// ---- HMI1/Screens/Motion/Mot_010_Motions.TcVIS
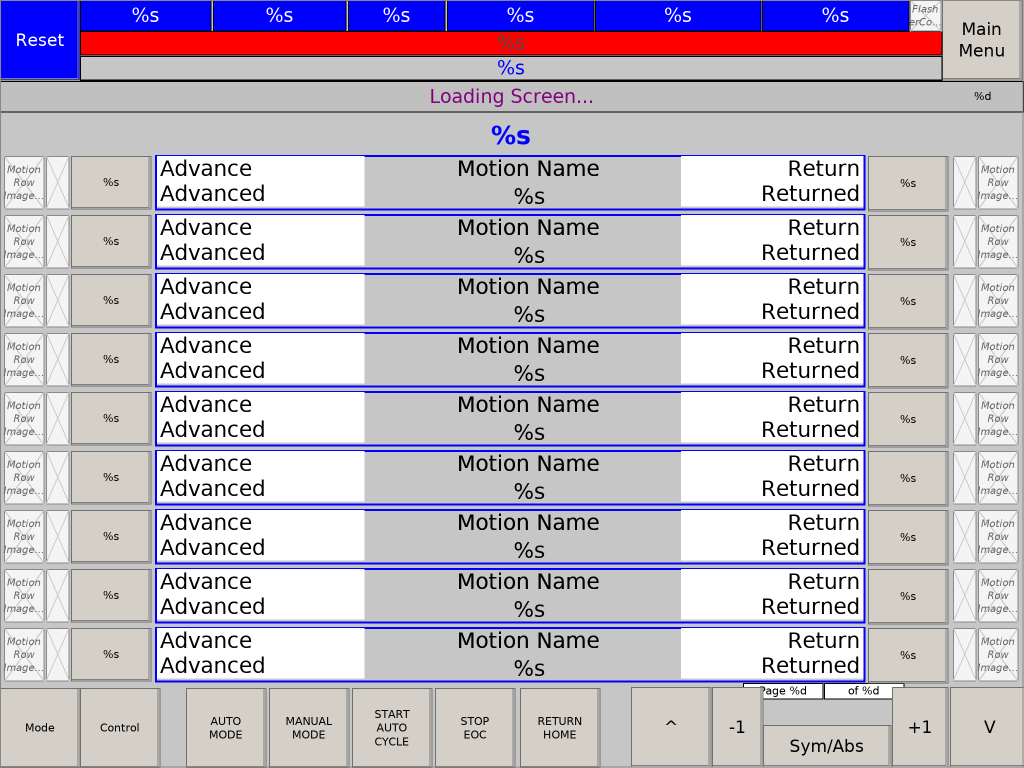
VISUALIZATION Mot_010_Motions  // 1024x768
    Frame (0,0 1024x768)
        shows Tmp_000_Template(header := gHMIData.hmiHeader)
    Frame (0,155 1024x55)
        shows MotionRow(MotionRowInstanceSingle := gHMIMotionRows.gMotionRows.gMotionRow1, MotionRowButtonsSingle := gHMIMotionRows.gMotionRowButtons.gMotionRow1btn)
    Frame (0,214 1024x55)
        shows MotionRow(MotionRowInstanceSingle := gHMIMotionRows.gMotionRows.gMotionRow2, MotionRowButtonsSingle := gHMIMotionRows.gMotionRowButtons.gMotionRow2btn)
    Frame (0,273 1024x55)
        shows MotionRow(MotionRowInstanceSingle := gHMIMotionRows.gMotionRows.gMotionRow3, MotionRowButtonsSingle := gHMIMotionRows.gMotionRowButtons.gMotionRow3btn)
    Frame (0,332 1024x55)
        shows MotionRow(MotionRowInstanceSingle := gHMIMotionRows.gMotionRows.gMotionRow4, MotionRowButtonsSingle := gHMIMotionRows.gMotionRowButtons.gMotionRow4btn)
    Frame (0,391 1024x55)
        shows MotionRow(MotionRowInstanceSingle := gHMIMotionRows.gMotionRows.gMotionRow5, MotionRowButtonsSingle := gHMIMotionRows.gMotionRowButtons.gMotionRow5btn)
    Frame (0,450 1024x55)
        shows MotionRow(MotionRowInstanceSingle := gHMIMotionRows.gMotionRows.gMotionRow6, MotionRowButtonsSingle := gHMIMotionRows.gMotionRowButtons.gMotionRow6btn)
    Button (763,725 128x42), "Sym/Abs", colour toggle: gHMIButtons.btnAbsMode
        toggle gHMIButtons.btnAbsMode
        OnMouseDown: execute { gHMIButtons.gAnyButtonPressed := TRUE; }
    Button (631,687 80x80), "^"
        tap gHMIButtons.btnPrevPage
        OnMouseDown: execute { gHMIButtons.gAnyButtonPressed := TRUE; }
    Button (950,687 80x80), "V"
        tap gHMIButtons.btnNextPage
        OnMouseDown: execute { gHMIButtons.gAnyButtonPressed := TRUE; }
    Rectangle (743,683 80x16), "Page %d", text variable: gHMIData.gActivePageNumber
        OnMouseDown: execute { gHMIButtons.gAnyButtonPressed := TRUE; }
    Rectangle (824,683 80x16), "of %d", text variable: gHMIData.gMaxPageNumber
        OnMouseDown: execute { gHMIButtons.gAnyButtonPressed := TRUE; }
    Rectangle (5,116 1012x38), "%s", text list: 'ManualPageTitle', text index: gHMIData.gManualScreenTitle
    Frame (0,509 1024x55)
        shows MotionRow(MotionRowInstanceSingle := gHMIMotionRows.gMotionRows.gMotionRow7, MotionRowButtonsSingle := gHMIMotionRows.gMotionRowButtons.gMotionRow7btn)
    Frame (0,568 1024x55)
        shows MotionRow(MotionRowInstanceSingle := gHMIMotionRows.gMotionRows.gMotionRow8, MotionRowButtonsSingle := gHMIMotionRows.gMotionRowButtons.gMotionRow8btn)
    Frame (0,627 1024x55)
        shows MotionRow(MotionRowInstanceSingle := gHMIMotionRows.gMotionRows.gMotionRow9, MotionRowButtonsSingle := gHMIMotionRows.gMotionRowButtons.gMotionRow9btn)
    Button (712,687 51x80), "-1"
        tap gHMIButtons.btnNeg1Row
        OnMouseDown: execute { gHMIButtons.gAnyButtonPressed := TRUE; }
    Button (892,687 56x80), "+1"
        tap gHMIButtons.btnPlus1Row
        OnMouseDown: execute { gHMIButtons.gAnyButtonPressed := TRUE; }
END_VISUALIZATION

// ---- HMI1/Screens/Motion/Mot_011_Axis.TcVIS
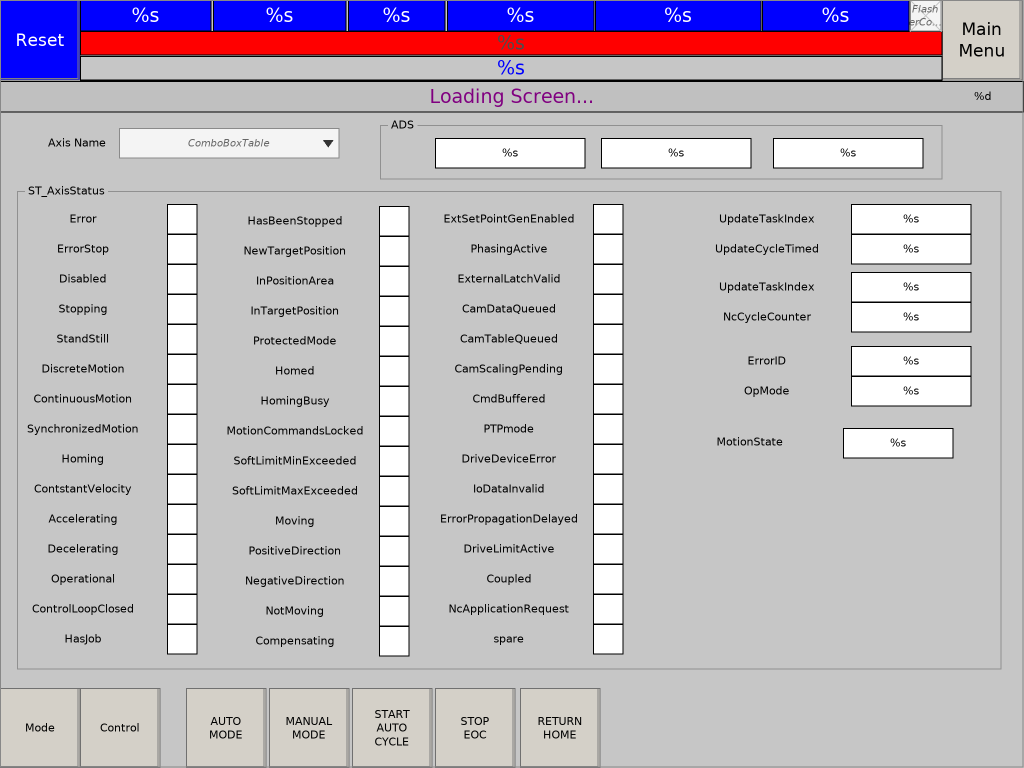
VISUALIZATION Mot_011_Axis  // 1024x768
    Frame (0,0 1024x768)
        shows Tmp_000_Template(header := gHMIData.hmiHeader)
    GroupBox (380,117 562x62), "ADS"
    GroupBox (17,183 984x486), "ST_AxisStatus"
        Label (658,244 150x30), "MotionState"
        Rectangle (826,245 110x30), "%s", text variable: driveGlobals.hmiAxis.Status.MotionState
    ComboBoxTable (119,128 220x30), variable: driveGlobals.hmiAxisSel, data array: driveGlobals.tAxisList
        p3854506369: driveGlobals.tAxisList[INDEX]
        p1128707560: Axis.gNumAxisInSystem
    Label (2,128 150x30), "Axis Name"
    Rectangle (435,138 150x30), "%s", text variable: driveGlobals.hmiAxis.ADS.Channel
    Rectangle (601,138 150x30), "%s", text variable: driveGlobals.hmiAxis.ADS.NetId
    Rectangle (773,138 150x30), "%s", text variable: driveGlobals.hmiAxis.ADS.Port
    Label (8,204 150x30), "Error"
    Rectangle (167,204 30x30), colour toggle: driveGlobals.hmiAxis.Status.Error
    Label (8,234 150x30), "ErrorStop"
    Rectangle (167,234 30x30), colour toggle: driveGlobals.hmiAxis.Status.ErrorStop
    Label (8,264 150x30), "Disabled"
    Rectangle (167,264 30x30), colour toggle: driveGlobals.hmiAxis.Status.Disabled
    Label (8,294 150x30), "Stopping"
    Rectangle (167,294 30x30), colour toggle: driveGlobals.hmiAxis.Status.Stopping
    Label (8,324 150x30), "StandStill"
    Rectangle (167,324 30x30), colour toggle: driveGlobals.hmiAxis.Status.StandStill
    Label (8,354 150x30), "DiscreteMotion"
    Rectangle (167,354 30x30), colour toggle: driveGlobals.hmiAxis.Status.DiscreteMotion
    Label (8,384 150x30), "ContinuousMotion"
    Rectangle (167,384 30x30), colour toggle: driveGlobals.hmiAxis.Status.ContinuousMotion
    Label (8,414 150x30), "SynchronizedMotion"
    Rectangle (167,414 30x30), colour toggle: driveGlobals.hmiAxis.Status.SynchronizedMotion
    Label (8,444 150x30), "Homing"
    Rectangle (167,444 30x30), colour toggle: driveGlobals.hmiAxis.Status.Homing
    Label (8,474 150x30), "ContstantVelocity"
    Rectangle (167,474 30x30), colour toggle: driveGlobals.hmiAxis.Status.ConstantVelocity
    Label (8,504 150x30), "Accelerating"
    Rectangle (167,504 30x30), colour toggle: driveGlobals.hmiAxis.Status.Accelerating
    Label (8,534 150x30), "Decelerating"
    Rectangle (167,534 30x30), colour toggle: driveGlobals.hmiAxis.Status.Decelerating
    Label (8,564 150x30), "Operational"
    Rectangle (167,564 30x30), colour toggle: driveGlobals.hmiAxis.Status.Operational
    Label (8,594 150x30), "ControlLoopClosed"
    Rectangle (167,594 30x30), colour toggle: driveGlobals.hmiAxis.Status.ControlLoopClosed
    Label (8,624 150x30), "HasJob"
    Rectangle (167,624 30x30), colour toggle: driveGlobals.hmiAxis.Status.HasJob
    Label (220,206 150x30), "HasBeenStopped"
    Rectangle (379,206 30x30), colour toggle: driveGlobals.hmiAxis.Status.HasBeenStopped
    Label (220,236 150x30), "NewTargetPosition"
    Rectangle (379,236 30x30), colour toggle: driveGlobals.hmiAxis.Status.NewTargetPosition
    Label (220,266 150x30), "InPositionArea"
    Rectangle (379,266 30x30), colour toggle: driveGlobals.hmiAxis.Status.InPositionArea
    Label (220,296 150x30), "InTargetPosition"
    Rectangle (379,296 30x30), colour toggle: driveGlobals.hmiAxis.Status.InTargetPosition
    Label (220,326 150x30), "ProtectedMode"
    Rectangle (379,326 30x30), colour toggle: driveGlobals.hmiAxis.Status.ProtectedMode
    Label (220,356 150x30), "Homed"
    Rectangle (379,356 30x30), colour toggle: driveGlobals.hmiAxis.Status.Homed
    Label (220,386 150x30), "HomingBusy"
    Rectangle (379,386 30x30), colour toggle: driveGlobals.hmiAxis.Status.HomingBusy
    Label (220,416 150x30), "MotionCommandsLocked"
    Rectangle (379,416 30x30), colour toggle: driveGlobals.hmiAxis.Status.MotionCommandsLocked
    Label (220,446 150x30), "SoftLimitMinExceeded"
    Rectangle (379,446 30x30), colour toggle: driveGlobals.hmiAxis.Status.SoftLimitMinExceeded
    Label (220,476 150x30), "SoftLimitMaxExceeded"
    Rectangle (379,476 30x30), colour toggle: driveGlobals.hmiAxis.Status.SoftLimitMaxExceeded
    Label (220,506 150x30), "Moving"
    Rectangle (379,506 30x30), colour toggle: driveGlobals.hmiAxis.Status.Moving
    Label (220,536 150x30), "PositiveDirection"
    Rectangle (379,536 30x30), colour toggle: driveGlobals.hmiAxis.Status.PositiveDirection
    Label (220,566 150x30), "NegativeDirection"
    Rectangle (379,566 30x30), colour toggle: driveGlobals.hmiAxis.Status.NegativeDirection
    Label (220,596 150x30), "NotMoving"
    Rectangle (379,596 30x30), colour toggle: driveGlobals.hmiAxis.Status.NotMoving
    Label (220,626 150x30), "Compensating"
    Rectangle (379,626 30x30), colour toggle: driveGlobals.hmiAxis.Status.Compensating
    Label (434,204 150x30), "ExtSetPointGenEnabled"
    Rectangle (593,204 30x30), colour toggle: driveGlobals.hmiAxis.Status.ExtSetPointGenEnabled
    Label (434,234 150x30), "PhasingActive"
    Rectangle (593,234 30x30), colour toggle: driveGlobals.hmiAxis.Status.PhasingActive
    Label (434,264 150x30), "ExternalLatchValid"
    Rectangle (593,264 30x30), colour toggle: driveGlobals.hmiAxis.Status.ExternalLatchValid
    Label (434,294 150x30), "CamDataQueued"
    Rectangle (593,294 30x30), colour toggle: driveGlobals.hmiAxis.Status.CamDataQueued
    Label (434,324 150x30), "CamTableQueued"
    Rectangle (593,324 30x30), colour toggle: driveGlobals.hmiAxis.Status.CamTableQueued
    Label (434,354 150x30), "CamScalingPending"
    Rectangle (593,354 30x30), colour toggle: driveGlobals.hmiAxis.Status.CamScalingPending
    Label (434,384 150x30), "CmdBuffered"
    Rectangle (593,384 30x30), colour toggle: driveGlobals.hmiAxis.Status.CmdBuffered
    Label (434,414 150x30), "PTPmode"
    Rectangle (593,414 30x30), colour toggle: driveGlobals.hmiAxis.Status.PTPmode
    Label (434,444 150x30), "DriveDeviceError"
    Rectangle (593,444 30x30), colour toggle: driveGlobals.hmiAxis.Status.DriveDeviceError
    Label (434,474 150x30), "IoDataInvalid"
    Rectangle (593,474 30x30), colour toggle: driveGlobals.hmiAxis.Status.IoDataInvalid
    Label (434,504 150x30), "ErrorPropagationDelayed"
    Rectangle (593,504 30x30), colour toggle: driveGlobals.hmiAxis.Status.ErrorPropagationDelayed
    Label (434,534 150x30), "DriveLimitActive"
    Rectangle (593,534 30x30), colour toggle: driveGlobals.hmiAxis.Status.DriveLimitActive
    Label (434,564 150x30), "Coupled"
    Rectangle (593,564 30x30), colour toggle: driveGlobals.hmiAxis.Status.Coupled
    Label (434,594 150x30), "NcApplicationRequest"
    Rectangle (593,594 30x30), colour toggle: driveGlobals.hmiAxis.Status.NcApplicationRequest
    Label (434,624 150x30), "spare"
    Rectangle (593,624 30x30)
    Label (692,204 150x30), "UpdateTaskIndex"
    Rectangle (851,204 120x30), "%s", text variable: driveGlobals.hmiAxis.Status.UpdateTaskIndex
    Label (692,234 150x30), "UpdateCycleTimed"
    Rectangle (851,234 120x30), "%s", text variable: driveGlobals.hmiAxis.Status.UpdateCycleTime
    Label (692,272 150x30), "UpdateTaskIndex"
    Rectangle (851,272 120x30), "%s"
    Label (692,302 150x30), "NcCycleCounter"
    Rectangle (851,302 120x30), "%s", text variable: driveGlobals.hmiAxis.Status.NcCycleCounter
    Label (692,346 150x30), "ErrorID"
    Rectangle (851,346 120x30), "%s", text variable: driveGlobals.hmiAxis.Status.ErrorID
    Label (692,376 150x30), "OpMode"
    Rectangle (851,376 120x30), "%s"
END_VISUALIZATION

// ---- HMI1/Screens/Popup/PopupMenu1.TcVIS
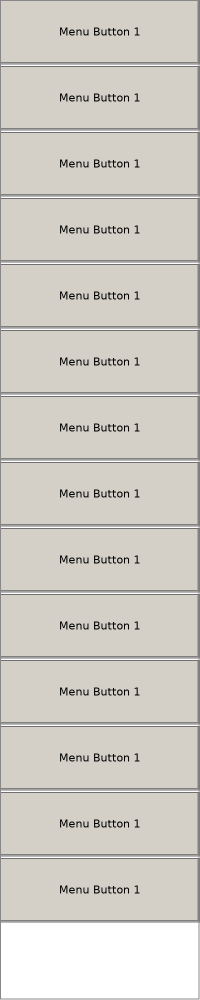
VISUALIZATION PopupMenu1  // 200x1000
    Button (0,0 200x64), "Menu Button 1"
    Button (0,66 200x64), "Menu Button 1"
    Button (0,132 200x64), "Menu Button 1"
    Button (0,198 200x64), "Menu Button 1"
    Button (0,264 200x64), "Menu Button 1"
    Button (0,330 200x64), "Menu Button 1"
    Button (0,396 200x64), "Menu Button 1"
    Button (0,462 200x64), "Menu Button 1"
    Button (0,528 200x64), "Menu Button 1"
    Button (0,594 200x64), "Menu Button 1"
    Button (0,660 200x64), "Menu Button 1"
    Button (0,726 200x64), "Menu Button 1"
    Button (0,792 200x64), "Menu Button 1"
    Button (0,858 200x64), "Menu Button 1"
END_VISUALIZATION

// ---- HMI1/Screens/Popup/PopupMenu2.TcVIS
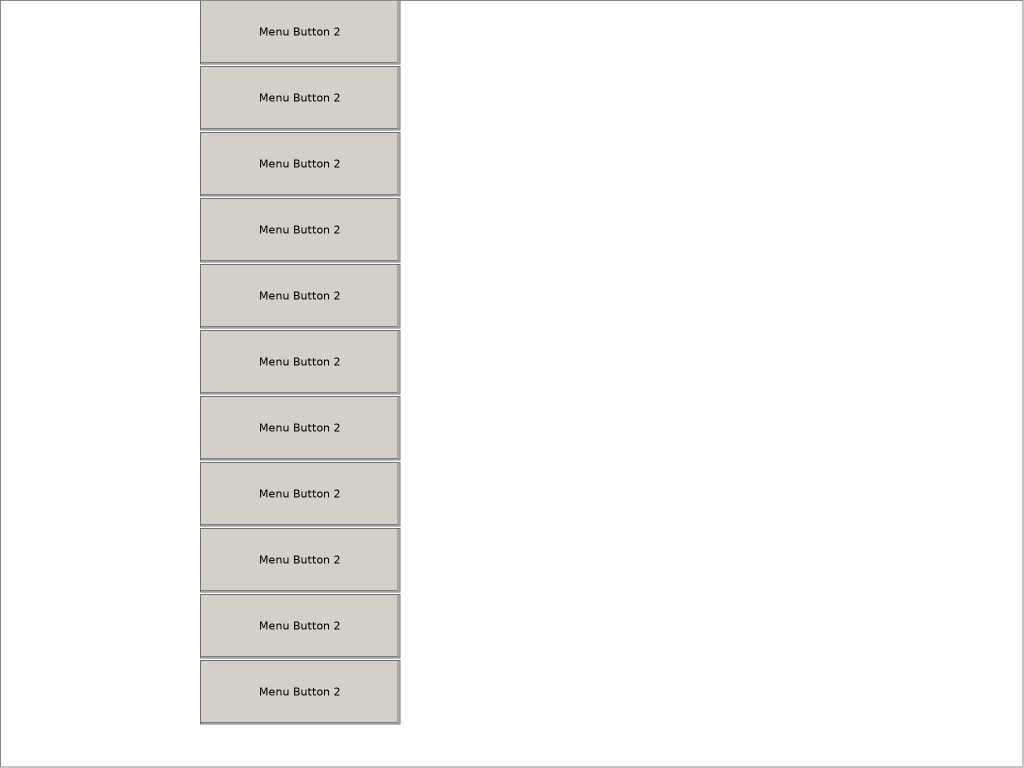
VISUALIZATION PopupMenu2  // 1024x768
    Button (200,0 200x64), "Menu Button 2"
        OnMouseClick: CloseDialog Dialog=PopupMenu2, Result=None, NumpadKeypadSet=True
    Button (200,66 200x64), "Menu Button 2"
        OnMouseClick: CloseDialog Dialog=PopupMenu2, Result=None, NumpadKeypadSet=True
    Button (200,132 200x64), "Menu Button 2"
        OnMouseClick: CloseDialog Dialog=PopupMenu2, Result=None, NumpadKeypadSet=True
    Button (200,198 200x64), "Menu Button 2"
        OnMouseClick: CloseDialog Dialog=PopupMenu2, Result=None, NumpadKeypadSet=True
    Button (200,264 200x64), "Menu Button 2"
        OnMouseClick: CloseDialog Dialog=PopupMenu2, Result=None, NumpadKeypadSet=True
    Button (200,330 200x64), "Menu Button 2"
        OnMouseClick: CloseDialog Dialog=PopupMenu2, Result=None, NumpadKeypadSet=True
    Button (200,396 200x64), "Menu Button 2"
        OnMouseClick: CloseDialog Dialog=PopupMenu2, Result=None, NumpadKeypadSet=True
    Button (200,462 200x64), "Menu Button 2"
        OnMouseClick: CloseDialog Dialog=PopupMenu2, Result=None, NumpadKeypadSet=True
    Button (200,528 200x64), "Menu Button 2"
        OnMouseClick: CloseDialog Dialog=PopupMenu2, Result=None, NumpadKeypadSet=True
    Button (200,594 200x64), "Menu Button 2"
        OnMouseClick: CloseDialog Dialog=PopupMenu2, Result=None, NumpadKeypadSet=True
    Button (200,660 200x64), "Menu Button 2"
        OnMouseClick: CloseDialog Dialog=PopupMenu2, Result=None, NumpadKeypadSet=True
    InvisibleInput (400,0 622x768)
        OnMouseClick: CloseDialog Dialog=PopupMenu2, Result=OK, NumpadKeypadSet=True
    InvisibleInput (0,0 200x768)
        OnMouseClick: CloseDialog Dialog=PopupMenu2, Result=OK, NumpadKeypadSet=True
    InvisibleInput (200,725 203x44)
        OnMouseClick: CloseDialog Dialog=PopupMenu2, Result=OK, NumpadKeypadSet=True
END_VISUALIZATION

// ---- HMI1/Screens/Popup/PopupMenu3.TcVIS
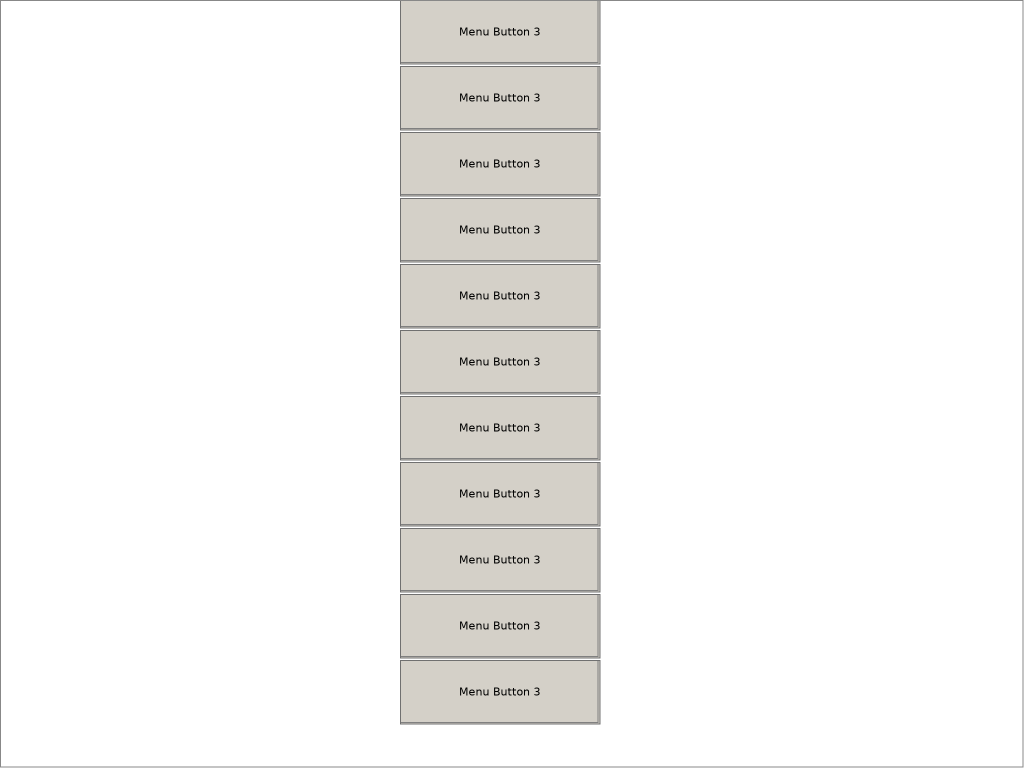
VISUALIZATION PopupMenu3  // 1024x768
    Button (400,0 200x64), "Menu Button 3"
        OnMouseClick: CloseDialog Dialog=PopupMenu3, Result=None, NumpadKeypadSet=True
    Button (400,66 200x64), "Menu Button 3"
        OnMouseClick: CloseDialog Dialog=PopupMenu3, Result=None, NumpadKeypadSet=True
    Button (400,132 200x64), "Menu Button 3"
        OnMouseClick: CloseDialog Dialog=PopupMenu3, Result=None, NumpadKeypadSet=True
    Button (400,198 200x64), "Menu Button 3"
        OnMouseClick: CloseDialog Dialog=PopupMenu3, Result=None, NumpadKeypadSet=True
    Button (400,264 200x64), "Menu Button 3"
        OnMouseClick: CloseDialog Dialog=PopupMenu3, Result=None, NumpadKeypadSet=True
    Button (400,330 200x64), "Menu Button 3"
        OnMouseClick: CloseDialog Dialog=PopupMenu3, Result=None, NumpadKeypadSet=True
    Button (400,396 200x64), "Menu Button 3"
        OnMouseClick: CloseDialog Dialog=PopupMenu3, Result=None, NumpadKeypadSet=True
    Button (400,462 200x64), "Menu Button 3"
        OnMouseClick: CloseDialog Dialog=PopupMenu3, Result=None, NumpadKeypadSet=True
    Button (400,528 200x64), "Menu Button 3"
        OnMouseClick: CloseDialog Dialog=PopupMenu3, Result=None, NumpadKeypadSet=True
    Button (400,594 200x64), "Menu Button 3"
        OnMouseClick: CloseDialog Dialog=PopupMenu3, Result=None, NumpadKeypadSet=True
    Button (400,660 200x64), "Menu Button 3"
        OnMouseClick: CloseDialog Dialog=PopupMenu3, Result=None, NumpadKeypadSet=True
    InvisibleInput (600,0 425x768)
        OnMouseClick: CloseDialog Dialog=PopupMenu3, Result=OK, NumpadKeypadSet=True
    InvisibleInput (0,0 400x768)
        OnMouseClick: CloseDialog Dialog=PopupMenu3, Result=OK, NumpadKeypadSet=True
    InvisibleInput (400,725 203x44)
        OnMouseClick: CloseDialog Dialog=PopupMenu3, Result=OK, NumpadKeypadSet=True
END_VISUALIZATION

// ---- HMI1/Screens/Popup/PopupMenu4.TcVIS
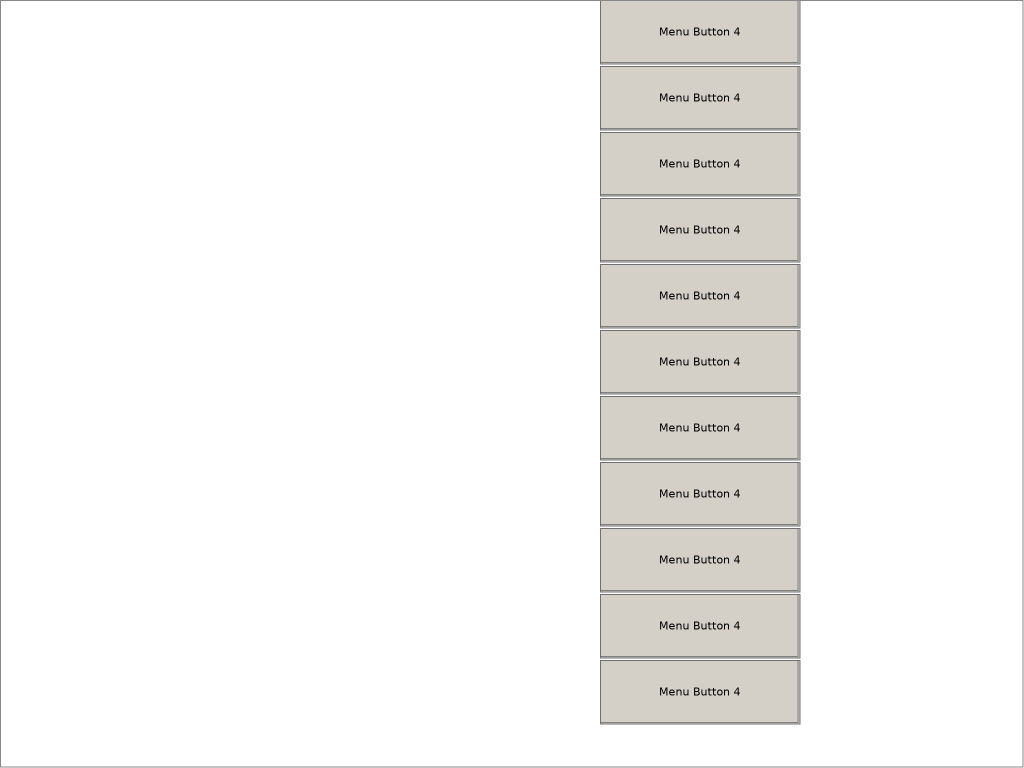
VISUALIZATION PopupMenu4  // 1024x768
    Button (600,0 200x64), "Menu Button 4"
        OnMouseClick: CloseDialog Dialog=PopupMenu4, Result=None, NumpadKeypadSet=True
    Button (600,66 200x64), "Menu Button 4"
        OnMouseClick: CloseDialog Dialog=PopupMenu4, Result=None, NumpadKeypadSet=True
    Button (600,132 200x64), "Menu Button 4"
        OnMouseClick: CloseDialog Dialog=PopupMenu4, Result=None, NumpadKeypadSet=True
    Button (600,198 200x64), "Menu Button 4"
        OnMouseClick: CloseDialog Dialog=PopupMenu4, Result=None, NumpadKeypadSet=True
    Button (600,264 200x64), "Menu Button 4"
        OnMouseClick: CloseDialog Dialog=PopupMenu4, Result=None, NumpadKeypadSet=True
    Button (600,330 200x64), "Menu Button 4"
        OnMouseClick: CloseDialog Dialog=PopupMenu4, Result=None, NumpadKeypadSet=True
    Button (600,396 200x64), "Menu Button 4"
        OnMouseClick: CloseDialog Dialog=PopupMenu4, Result=None, NumpadKeypadSet=True
    Button (600,462 200x64), "Menu Button 4"
        OnMouseClick: CloseDialog Dialog=PopupMenu4, Result=None, NumpadKeypadSet=True
    Button (600,528 200x64), "Menu Button 4"
        OnMouseClick: CloseDialog Dialog=PopupMenu4, Result=None, NumpadKeypadSet=True
    Button (600,594 200x64), "Menu Button 4"
        OnMouseClick: CloseDialog Dialog=PopupMenu4, Result=None, NumpadKeypadSet=True
    Button (600,660 200x64), "Menu Button 4"
        OnMouseClick: CloseDialog Dialog=PopupMenu4, Result=None, NumpadKeypadSet=True
    InvisibleInput (800,0 227x768)
        OnMouseClick: CloseDialog Dialog=PopupMenu4, Result=OK, NumpadKeypadSet=True
    InvisibleInput (0,0 600x768)
        OnMouseClick: CloseDialog Dialog=PopupMenu4, Result=OK, NumpadKeypadSet=True
    InvisibleInput (600,725 203x44)
        OnMouseClick: CloseDialog Dialog=PopupMenu4, Result=OK, NumpadKeypadSet=True
END_VISUALIZATION

// ---- HMI1/Screens/Popup/PopupMenu5.TcVIS
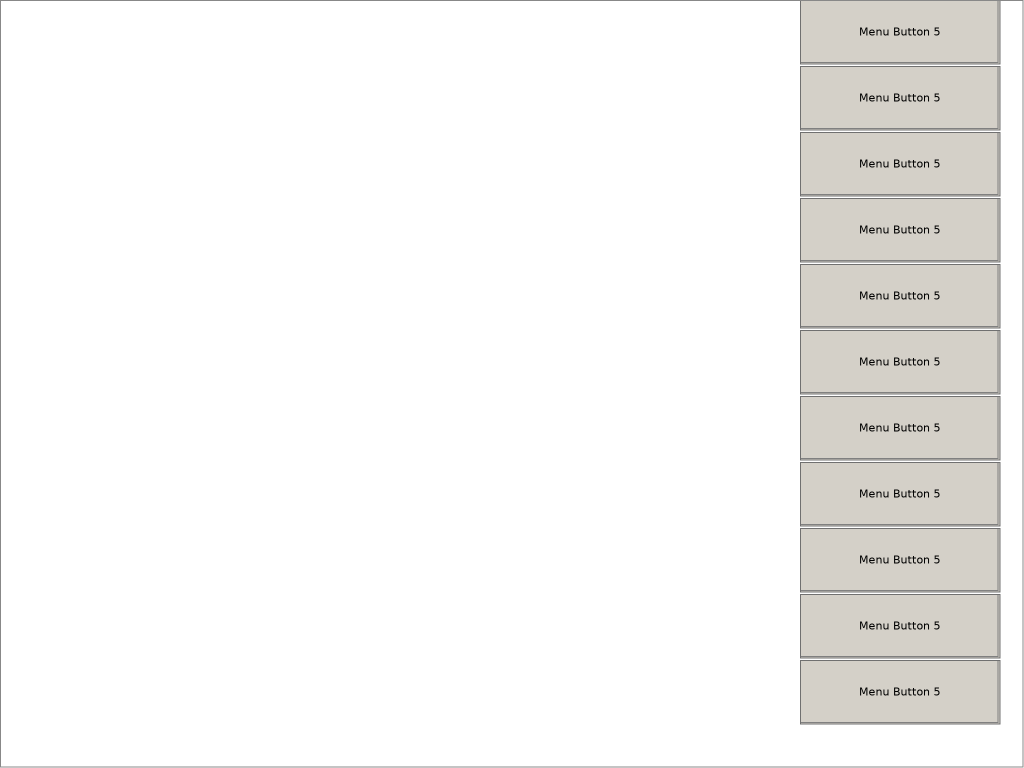
VISUALIZATION PopupMenu5  // 1024x768
    Button (800,0 200x64), "Menu Button 5"
        OnMouseClick: CloseDialog Dialog=PopupMenu5, Result=None, NumpadKeypadSet=True
    Button (800,66 200x64), "Menu Button 5"
        OnMouseClick: CloseDialog Dialog=PopupMenu5, Result=None, NumpadKeypadSet=True
    Button (800,132 200x64), "Menu Button 5"
        OnMouseClick: CloseDialog Dialog=PopupMenu5, Result=None, NumpadKeypadSet=True
    Button (800,198 200x64), "Menu Button 5"
        OnMouseClick: CloseDialog Dialog=PopupMenu5, Result=None, NumpadKeypadSet=True
    Button (800,264 200x64), "Menu Button 5"
        OnMouseClick: CloseDialog Dialog=PopupMenu5, Result=None, NumpadKeypadSet=True
    Button (800,330 200x64), "Menu Button 5"
        OnMouseClick: CloseDialog Dialog=PopupMenu5, Result=None, NumpadKeypadSet=True
    Button (800,396 200x64), "Menu Button 5"
        OnMouseClick: CloseDialog Dialog=PopupMenu5, Result=None, NumpadKeypadSet=True
    Button (800,462 200x64), "Menu Button 5"
        OnMouseClick: CloseDialog Dialog=PopupMenu5, Result=None, NumpadKeypadSet=True
    Button (800,528 200x64), "Menu Button 5"
        OnMouseClick: CloseDialog Dialog=PopupMenu5, Result=None, NumpadKeypadSet=True
    Button (800,594 200x64), "Menu Button 5"
        OnMouseClick: CloseDialog Dialog=PopupMenu5, Result=None, NumpadKeypadSet=True
    Button (800,660 200x64), "Menu Button 5"
        OnMouseClick: CloseDialog Dialog=PopupMenu5, Result=None, NumpadKeypadSet=True
    InvisibleInput (1000,0 25x768)
        OnMouseClick: CloseDialog Dialog=PopupMenu5, Result=Cancel, NumpadKeypadSet=True
    InvisibleInput (0,0 800x768)
        OnMouseClick: CloseDialog Dialog=PopupMenu5, Result=OK, NumpadKeypadSet=True
    InvisibleInput (800,726 203x44)
        OnMouseClick: CloseDialog Dialog=PopupMenu5, Result=Cancel, NumpadKeypadSet=True
END_VISUALIZATION

// ---- HMI1/Templates/AxisRow.TcVIS
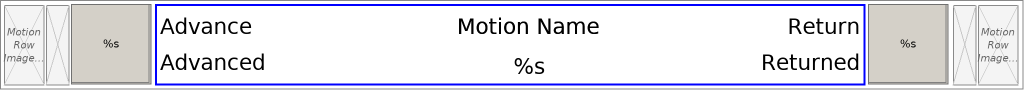
VISUALIZATION AxisRow  // 1024x90
VAR_IN_OUT
	MotionRowInstanceSingle:typeMotionRow; //feedback to motion row to operator
	MotionRowButtonsSingle:typeMotionRowButtons; //button feedback in seperate interface
END_VAR
    Rectangle (155,4 710x81), invisible if: MotionRowInstanceSingle.Returned.bHideCoil AND MotionRowInstanceSingle.bHideName
    Button (868,4 80x80), "%s", text variable: MotionRowInstanceSingle.Returned.NumberOrder, invisible if: MotionRowInstanceSingle.Returned.bHideButton
        tap MotionRowButtonsSingle.btnReturn
        OnMouseDown: execute { gHMIButtons.gAnyButtonPressed := TRUE; }
    Button (71,4 80x80), "%s", text variable: MotionRowInstanceSingle.Advance.NumberOrder, invisible if: MotionRowInstanceSingle.Advance.bHideButton
        tap MotionRowButtonsSingle.btnAdvance
        OnMouseDown: execute { gHMIButtons.gAnyButtonPressed := TRUE; }
    Rectangle (393,50 273x33), "%s", text variable: MotionRowInstanceSingle.strPosn, invisible if: MotionRowInstanceSingle.bHidePosn
    Group (157,10 706x69)
        Rectangle (524,0 182x33), "Return", invisible if: MotionRowInstanceSingle.Returned.bHideCoil or MotionRowInstanceSingle.bIsAbsSymSwitch, text list: 'AxisRowText', text index: MotionRowInstanceSingle.IndexLocation + 3, colour variable: MotionRowInstanceSingle.Returned.CoilColour
        Rectangle (235,0 273x33), "Motion Name", invisible if: MotionRowInstanceSingle.bHideName or MotionRowInstanceSingle.bIsAbsSymSwitch, text list: 'AxisRowText', text index: MotionRowInstanceSingle.IndexLocation + 6
        Rectangle (524,36 182x33), "Returned", invisible if: MotionRowInstanceSingle.Returned.bHideDepth or MotionRowInstanceSingle.bIsAbsSymSwitch, text list: 'AxisRowText', text index: MotionRowInstanceSingle.IndexLocation + 4, colour variable: MotionRowInstanceSingle.Returned.FdbkColour
        Rectangle (0,0 207x33), "Advance", text variable: MotionRowInstanceSingle.Advance.valCoil, invisible if: MotionRowInstanceSingle.Advance.bHideCoil or MotionRowInstanceSingle.bIsAbsSymSwitch, text list: 'AxisRowText', text index: MotionRowInstanceSingle.IndexLocation + 0, colour variable: MotionRowInstanceSingle.Advance.CoilColour
        Rectangle (0,36 207x33), "Advanced", invisible if: MotionRowInstanceSingle.Advance.bHideDepth or MotionRowInstanceSingle.bIsAbsSymSwitch, text list: 'AxisRowText', text index: MotionRowInstanceSingle.IndexLocation + 1, colour variable: MotionRowInstanceSingle.Advance.FdbkColour
    Image (4,5 40x80), invisible if: NOT MotionRowInstanceSingle.Advance.InterlockOK OR MotionRowInstanceSingle.Advance.bHideInterlock, image: MotionRowImages.LeftHighlight
    Image (4,5 40x80), invisible if: MotionRowInstanceSingle.Advance.InterlockOK OR MotionRowInstanceSingle.Advance.bHideInterlock, image: MotionRowImages.LeftNot
    Image (978,5 40x80), invisible if: MotionRowInstanceSingle.Returned.InterlockOK OR MotionRowInstanceSingle.Returned.bHideInterlock, image: MotionRowImages.RightNot
    Image (978,5 40x80), invisible if: NOT MotionRowInstanceSingle.Returned.InterlockOK OR MotionRowInstanceSingle.Returned.bHideInterlock, image: MotionRowImages.RightHighlight
    Image (46,5 23x80), invisible if: MotionRowInstanceSingle.Advance.Prompt OR MotionRowInstanceSingle.Advance.bHidePrompt, image: MotionRowImages.PromptNOK
    Image (953,5 23x80), invisible if: NOT MotionRowInstanceSingle.Returned.Prompt OR MotionRowInstanceSingle.Returned.bHidePrompt, image: MotionRowImages.PromptOK
    Image (953,5 23x80), invisible if: MotionRowInstanceSingle.Returned.Prompt OR MotionRowInstanceSingle.Returned.bHidePrompt, image: MotionRowImages.PromptNOK
    Image (46,5 23x80), invisible if: NOT MotionRowInstanceSingle.Advance.Prompt OR MotionRowInstanceSingle.Advance.bHidePrompt, image: MotionRowImages.PromptOK
    Group (157,10 706x69)
        Rectangle (524,0 182x33), "Return", invisible if: MotionRowInstanceSingle.Returned.bHideCoil or NOT MotionRowInstanceSingle.bIsAbsSymSwitch, text list: 'AxisRowText', text index: MotionRowInstanceSingle.IndexLocation + 3 + 10, colour variable: MotionRowInstanceSingle.Returned.CoilColour
        Rectangle (235,0 273x33), "Motion Name", invisible if: MotionRowInstanceSingle.bHideName or NOT MotionRowInstanceSingle.bIsAbsSymSwitch, text list: 'AxisRowText', text index: MotionRowInstanceSingle.IndexLocation + 6 + 10
        Rectangle (524,36 182x33), "Returned", invisible if: MotionRowInstanceSingle.Returned.bHideDepth or NOT MotionRowInstanceSingle.bIsAbsSymSwitch, text list: 'AxisRowText', text index: MotionRowInstanceSingle.IndexLocation + 4 + 10, colour variable: MotionRowInstanceSingle.Returned.FdbkColour
        Rectangle (0,0 207x33), "Advance", text variable: MotionRowInstanceSingle.Advance.valCoil, invisible if: MotionRowInstanceSingle.Advance.bHideCoil or NOT MotionRowInstanceSingle.bIsAbsSymSwitch, text list: 'AxisRowText', text index: MotionRowInstanceSingle.IndexLocation + 0 + 10, colour variable: MotionRowInstanceSingle.Advance.CoilColour
        Rectangle (0,36 207x33), "Advanced", invisible if: MotionRowInstanceSingle.Advance.bHideDepth or NOT MotionRowInstanceSingle.bIsAbsSymSwitch, text list: 'AxisRowText', text index: MotionRowInstanceSingle.IndexLocation + 1 + 10, colour variable: MotionRowInstanceSingle.Advance.FdbkColour
END_VISUALIZATION

// ---- HMI1/Templates/LanguageRow.TcVIS
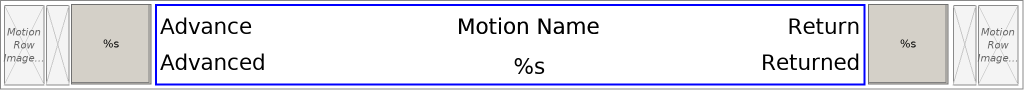
VISUALIZATION LanguageRow  // 1024x90
VAR_IN_OUT
	MotionRowInstanceSingle:typeMotionRow; //feedback to motion row to operator
	MotionRowButtonsSingle:typeMotionRowButtons; //button feedback in seperate interface
END_VAR
    Rectangle (155,4 710x81), invisible if: MotionRowInstanceSingle.Returned.bHideCoil AND MotionRowInstanceSingle.bHideName
    Button (868,4 80x80), "%s", text variable: MotionRowInstanceSingle.Returned.NumberOrder, invisible if: MotionRowInstanceSingle.Returned.bHideButton
        tap MotionRowButtonsSingle.btnReturn
        OnMouseDown: execute { gHMIButtons.gAnyButtonPressed := TRUE; }
    Button (71,4 80x80), "%s", text variable: MotionRowInstanceSingle.Advance.NumberOrder, invisible if: MotionRowInstanceSingle.Advance.bHideButton
        tap MotionRowButtonsSingle.btnAdvance
        OnMouseDown: execute { gHMIButtons.gAnyButtonPressed := TRUE; }
    Rectangle (393,50 273x33), "%s", text variable: MotionRowInstanceSingle.strPosn, invisible if: MotionRowInstanceSingle.bHidePosn
    Group (157,10 706x69)
        Rectangle (524,0 182x33), "Return", invisible if: MotionRowInstanceSingle.Returned.bHideCoil or MotionRowInstanceSingle.bIsAbsSymSwitch, text list: 'LanguageRowText', text index: MotionRowInstanceSingle.IndexLocation + 3, colour variable: MotionRowInstanceSingle.Returned.CoilColour
        Rectangle (235,0 273x33), "Motion Name", invisible if: MotionRowInstanceSingle.bHideName or MotionRowInstanceSingle.bIsAbsSymSwitch, text list: 'LanguageRowText', text index: MotionRowInstanceSingle.IndexLocation + 6
        Rectangle (524,36 182x33), "Returned", invisible if: MotionRowInstanceSingle.Returned.bHideDepth or MotionRowInstanceSingle.bIsAbsSymSwitch, text list: 'LanguageRowText', text index: MotionRowInstanceSingle.IndexLocation + 4, colour variable: MotionRowInstanceSingle.Returned.FdbkColour
        Rectangle (0,0 207x33), "Advance", text variable: MotionRowInstanceSingle.Advance.valCoil, invisible if: MotionRowInstanceSingle.Advance.bHideCoil or MotionRowInstanceSingle.bIsAbsSymSwitch, text list: 'LanguageRowText', text index: MotionRowInstanceSingle.IndexLocation + 0, colour variable: MotionRowInstanceSingle.Advance.CoilColour
        Rectangle (0,36 207x33), "Advanced", invisible if: MotionRowInstanceSingle.Advance.bHideDepth or MotionRowInstanceSingle.bIsAbsSymSwitch, text list: 'LanguageRowText', text index: MotionRowInstanceSingle.IndexLocation + 1, colour variable: MotionRowInstanceSingle.Advance.FdbkColour
    Image (4,5 40x80), invisible if: NOT MotionRowInstanceSingle.Advance.InterlockOK OR MotionRowInstanceSingle.Advance.bHideInterlock, image: MotionRowImages.LeftHighlight
    Image (4,5 40x80), invisible if: MotionRowInstanceSingle.Advance.InterlockOK OR MotionRowInstanceSingle.Advance.bHideInterlock, image: MotionRowImages.LeftNot
    Image (978,5 40x80), invisible if: MotionRowInstanceSingle.Returned.InterlockOK OR MotionRowInstanceSingle.Returned.bHideInterlock, image: MotionRowImages.RightNot
    Image (978,5 40x80), invisible if: NOT MotionRowInstanceSingle.Returned.InterlockOK OR MotionRowInstanceSingle.Returned.bHideInterlock, image: MotionRowImages.RightHighlight
    Image (46,5 23x80), invisible if: MotionRowInstanceSingle.Advance.Prompt OR MotionRowInstanceSingle.Advance.bHidePrompt, image: MotionRowImages.PromptNOK
    Image (953,5 23x80), invisible if: NOT MotionRowInstanceSingle.Returned.Prompt OR MotionRowInstanceSingle.Returned.bHidePrompt, image: MotionRowImages.PromptOK
    Image (953,5 23x80), invisible if: MotionRowInstanceSingle.Returned.Prompt OR MotionRowInstanceSingle.Returned.bHidePrompt, image: MotionRowImages.PromptNOK
    Image (46,5 23x80), invisible if: NOT MotionRowInstanceSingle.Advance.Prompt OR MotionRowInstanceSingle.Advance.bHidePrompt, image: MotionRowImages.PromptOK
    Group (157,10 706x69)
        Rectangle (524,0 182x33), "Return", invisible if: MotionRowInstanceSingle.Returned.bHideCoil or NOT MotionRowInstanceSingle.bIsAbsSymSwitch, text list: 'LanguageRowText', text index: MotionRowInstanceSingle.IndexLocation + 3 + 10, colour variable: MotionRowInstanceSingle.Returned.CoilColour
        Rectangle (235,0 273x33), "Motion Name", invisible if: MotionRowInstanceSingle.bHideName or NOT MotionRowInstanceSingle.bIsAbsSymSwitch, text list: 'LanguageRowText', text index: MotionRowInstanceSingle.IndexLocation + 6 + 10
        Rectangle (524,36 182x33), "Returned", invisible if: MotionRowInstanceSingle.Returned.bHideDepth or NOT MotionRowInstanceSingle.bIsAbsSymSwitch, text list: 'LanguageRowText', text index: MotionRowInstanceSingle.IndexLocation + 4 + 10, colour variable: MotionRowInstanceSingle.Returned.FdbkColour
        Rectangle (0,0 207x33), "Advance", text variable: MotionRowInstanceSingle.Advance.valCoil, invisible if: MotionRowInstanceSingle.Advance.bHideCoil or NOT MotionRowInstanceSingle.bIsAbsSymSwitch, text list: 'LanguageRowText', text index: MotionRowInstanceSingle.IndexLocation + 0 + 10, colour variable: MotionRowInstanceSingle.Advance.CoilColour
        Rectangle (0,36 207x33), "Advanced", invisible if: MotionRowInstanceSingle.Advance.bHideDepth or NOT MotionRowInstanceSingle.bIsAbsSymSwitch, text list: 'LanguageRowText', text index: MotionRowInstanceSingle.IndexLocation + 1 + 10, colour variable: MotionRowInstanceSingle.Advance.FdbkColour
END_VISUALIZATION

// ---- HMI1/Templates/ModeRow.TcVIS
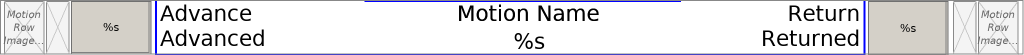
VISUALIZATION ModeRow  // 1024x55
VAR_IN_OUT
	MotionRowInstanceSingle:typeMotionRow; //feedback to motion row to operator
	MotionRowButtonsSingle:typeMotionRowButtons; //button feedback in seperate interface
END_VAR
    Rectangle (155,0 710x55), invisible if: MotionRowInstanceSingle.Returned.bHideCoil AND MotionRowInstanceSingle.bHideName
    Button (868,1 80x55), "%s", text variable: MotionRowInstanceSingle.Returned.NumberOrder, invisible if: MotionRowInstanceSingle.Returned.bHideButton
        tap MotionRowButtonsSingle.btnReturn
        OnMouseDown: execute { gHMIButtons.gAnyButtonPressed := TRUE; }
    Button (71,1 80x53), "%s", text variable: MotionRowInstanceSingle.Advance.NumberOrder, invisible if: MotionRowInstanceSingle.Advance.bHideButton
        tap MotionRowButtonsSingle.btnAdvance
        OnMouseDown: execute { gHMIButtons.gAnyButtonPressed := TRUE; }
    Rectangle (393,25 273x33), "%s", text variable: MotionRowInstanceSingle.strPosn, invisible if: MotionRowInstanceSingle.bHidePosn
    Group (157,1 706x52)
        Rectangle (524,0 182x25), "Return", invisible if: MotionRowInstanceSingle.Returned.bHideCoil or MotionRowInstanceSingle.bIsAbsSymSwitch, text list: 'ModeRowText', text index: MotionRowInstanceSingle.IndexLocation + 3, colour variable: MotionRowInstanceSingle.Returned.CoilColour
        Rectangle (235,0 273x25), "Motion Name", invisible if: MotionRowInstanceSingle.bHideName or MotionRowInstanceSingle.bIsAbsSymSwitch, text list: 'ModeRowText', text index: MotionRowInstanceSingle.IndexLocation + 6
        Rectangle (524,25 182x25), "Returned", invisible if: MotionRowInstanceSingle.Returned.bHideDepth or MotionRowInstanceSingle.bIsAbsSymSwitch, text list: 'ModeRowText', text index: MotionRowInstanceSingle.IndexLocation + 4, colour variable: MotionRowInstanceSingle.Returned.FdbkColour
        Rectangle (0,0 207x25), "Advance", text variable: MotionRowInstanceSingle.Advance.valCoil, invisible if: MotionRowInstanceSingle.Advance.bHideCoil or MotionRowInstanceSingle.bIsAbsSymSwitch, text list: 'ModeRowText', text index: MotionRowInstanceSingle.IndexLocation + 0, colour variable: MotionRowInstanceSingle.Advance.CoilColour
        Rectangle (0,25 207x25), "Advanced", invisible if: MotionRowInstanceSingle.Advance.bHideDepth or MotionRowInstanceSingle.bIsAbsSymSwitch, text list: 'ModeRowText', text index: MotionRowInstanceSingle.IndexLocation + 1, colour variable: MotionRowInstanceSingle.Advance.FdbkColour
    Image (4,1 40x53), invisible if: NOT MotionRowInstanceSingle.Advance.InterlockOK OR MotionRowInstanceSingle.Advance.bHideInterlock, image: MotionRowImages.LeftHighlight
    Image (4,1 40x53), invisible if: MotionRowInstanceSingle.Advance.InterlockOK OR MotionRowInstanceSingle.Advance.bHideInterlock, image: MotionRowImages.LeftNot
    Image (978,1 40x53), invisible if: MotionRowInstanceSingle.Returned.InterlockOK OR MotionRowInstanceSingle.Returned.bHideInterlock, image: MotionRowImages.RightNot
    Image (978,1 40x53), invisible if: NOT MotionRowInstanceSingle.Returned.InterlockOK OR MotionRowInstanceSingle.Returned.bHideInterlock, image: MotionRowImages.RightHighlight
    Image (46,1 23x53), invisible if: MotionRowInstanceSingle.Advance.Prompt OR MotionRowInstanceSingle.Advance.bHidePrompt, image: MotionRowImages.PromptNOK
    Image (953,1 23x53), invisible if: NOT MotionRowInstanceSingle.Returned.Prompt OR MotionRowInstanceSingle.Returned.bHidePrompt, image: MotionRowImages.PromptOK
    Image (953,1 23x53), invisible if: MotionRowInstanceSingle.Returned.Prompt OR MotionRowInstanceSingle.Returned.bHidePrompt, image: MotionRowImages.PromptNOK
    Image (46,1 23x53), invisible if: NOT MotionRowInstanceSingle.Advance.Prompt OR MotionRowInstanceSingle.Advance.bHidePrompt, image: MotionRowImages.PromptOK
    Group (157,1 706x52)
        Rectangle (524,0 182x25), "Return", invisible if: MotionRowInstanceSingle.Returned.bHideCoil or NOT MotionRowInstanceSingle.bIsAbsSymSwitch, text list: 'ModeRowText', text index: MotionRowInstanceSingle.IndexLocation + 3 + 10, colour variable: MotionRowInstanceSingle.Returned.CoilColour
        Rectangle (235,0 273x25), "Motion Name", invisible if: MotionRowInstanceSingle.bHideName or NOT MotionRowInstanceSingle.bIsAbsSymSwitch, text list: 'ModeRowText', text index: MotionRowInstanceSingle.IndexLocation + 6 + 10
        Rectangle (524,25 182x25), "Returned", invisible if: MotionRowInstanceSingle.Returned.bHideDepth or NOT MotionRowInstanceSingle.bIsAbsSymSwitch, text list: 'ModeRowText', text index: MotionRowInstanceSingle.IndexLocation + 4 + 10, colour variable: MotionRowInstanceSingle.Returned.FdbkColour
        Rectangle (0,0 207x25), "Advance", text variable: MotionRowInstanceSingle.Advance.valCoil, invisible if: MotionRowInstanceSingle.Advance.bHideCoil or NOT MotionRowInstanceSingle.bIsAbsSymSwitch, text list: 'ModeRowText', text index: MotionRowInstanceSingle.IndexLocation + 0 + 10, colour variable: MotionRowInstanceSingle.Advance.CoilColour
        Rectangle (0,25 207x25), "Advanced", invisible if: MotionRowInstanceSingle.Advance.bHideDepth or NOT MotionRowInstanceSingle.bIsAbsSymSwitch, text list: 'ModeRowText', text index: MotionRowInstanceSingle.IndexLocation + 1 + 10, colour variable: MotionRowInstanceSingle.Advance.FdbkColour
END_VISUALIZATION

// ---- HMI1/Templates/Tmp_001_Template_Alternate.TcVIS
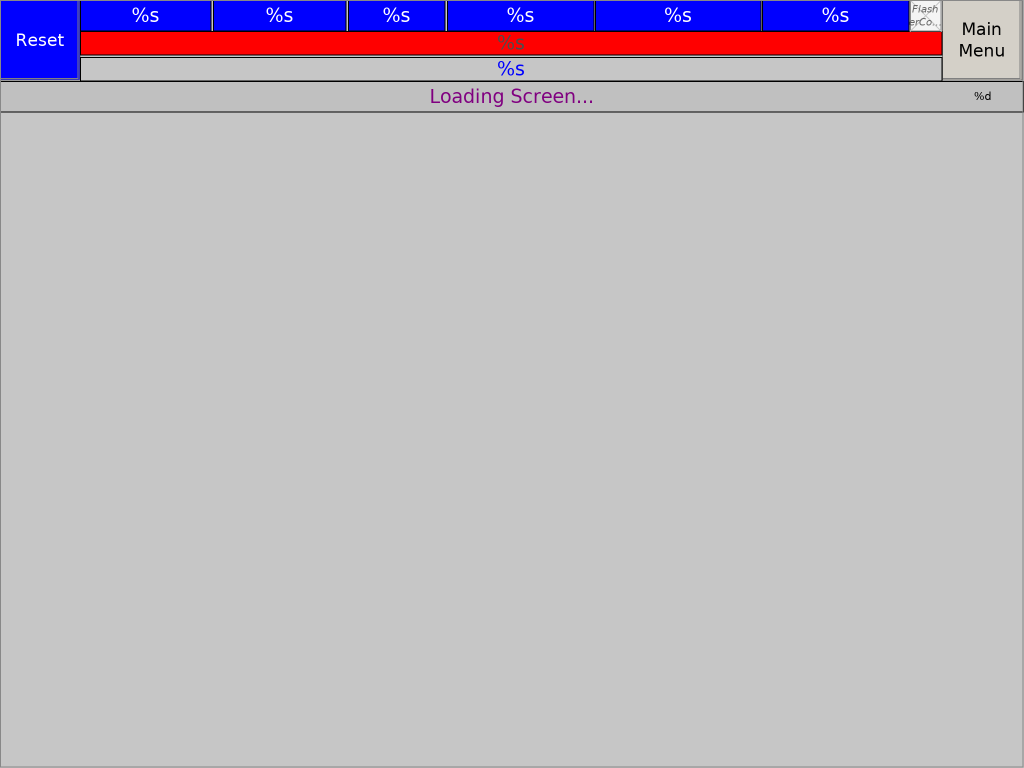
VISUALIZATION Tmp_001_Template_Alternate  // 1024x768
VAR_IN_OUT
	header:typeHMIheader;
	
END_VAR
    Rectangle (595,0 166x31)
        p2167032090: header.AnyStationWarningColour
    Rectangle (80,57 862x24)
    Group (0,0 1022x80)
        Button (0,0 80x80), "Reset"
            tap gHMIButtons.btnReset
            OnMouseDown: execute { gHMIButtons.gAnyButtonPressed := TRUE; }
        Button (942,0 80x80), "Main Menu"
            OnMouseClick: change screen: Men_030_MenuScreen
            OnMouseDown: execute { gHMIButtons.gAnyButtonPressed := TRUE; }
    Group (80,31 862x24)
        Rectangle (0,0 862x24), "%s", text variable: GlobalMessages.gMsgMc.Warning.topMessage, invisible if: gHMIData.gHideDisplayElementWarningView.McEnabled
        Rectangle (0,0 862x24), "%s", text variable: GlobalMessages.gMsgS1.Warning.topMessage, invisible if: gHMIData.gHideDisplayElementWarningView.S1Enabled
        Rectangle (0,0 862x24), "%s", text variable: GlobalMessages.gMsgS2.Warning.topMessage, invisible if: gHMIData.gHideDisplayElementWarningView.S2Enabled
        Rectangle (0,0 862x24), "%s", text variable: GlobalMessages.gMsgS3.Warning.topMessage, invisible if: gHMIData.gHideDisplayElementWarningView.S3Enabled
        Rectangle (0,0 862x24), "%s", text variable: GlobalMessages.gMsgS4.Warning.topMessage, invisible if: gHMIData.gHideDisplayElementWarningView.S4Enabled
        Rectangle (0,0 862x24), "%s", text variable: GlobalMessages.gMsgS5.Warning.topMessage, invisible if: gHMIData.gHideDisplayElementWarningView.S5Enabled
        Rectangle (0,0 862x24), "%s", text variable: GlobalMessages.gMsgS6.Warning.topMessage, invisible if: gHMIData.gHideDisplayElementWarningView.S6Enabled
    Group (80,31 862x24)
        OnMouseClick: change screen: Msg_020_Alarms
        Rectangle (0,0 862x24), "%s", text variable: GlobalMessages.gMsgMc.Alarm.topMessage, invisible if: gHMIData.gHideDisplayElementAlarmView.McEnabled
        Rectangle (0,0 862x24), "%s", text variable: GlobalMessages.gMsgS1.Alarm.topMessage, invisible if: gHMIData.gHideDisplayElementAlarmView.S1Enabled, text list: ''
        Rectangle (0,0 862x24), "%s", text variable: GlobalMessages.gMsgS2.Alarm.topMessage, invisible if: gHMIData.gHideDisplayElementAlarmView.S2Enabled
        Rectangle (0,0 862x24), "%s", text variable: GlobalMessages.gMsgS3.Alarm.topMessage, invisible if: gHMIData.gHideDisplayElementAlarmView.S3Enabled
        Rectangle (0,0 862x24), "%s", text variable: GlobalMessages.gMsgS4.Alarm.topMessage, invisible if: gHMIData.gHideDisplayElementAlarmView.S4Enabled
        Rectangle (0,0 862x24), "%s", text variable: GlobalMessages.gMsgS5.Alarm.topMessage, invisible if: gHMIData.gHideDisplayElementAlarmView.S5Enabled
        Rectangle (0,0 862x24), "%s", text variable: GlobalMessages.gMsgS6.Alarm.topMessage, invisible if: gHMIData.gHideDisplayElementAlarmView.S6Enabled
    Group (80,57 862x24)
        Rectangle (0,0 862x24), "%s", text variable: GlobalMessages.gMsgMc.Prompts.topMessage, invisible if: gHMIData.gHideDisplayElementPromptView.McEnabled
        Rectangle (0,0 862x24), "%s", text variable: GlobalMessages.gMsgS1.Prompts.topMessage, invisible if: gHMIData.gHideDisplayElementPromptView.S1Enabled
        Rectangle (0,0 862x24), "%s", text variable: GlobalMessages.gMsgS2.Prompts.topMessage, invisible if: gHMIData.gHideDisplayElementPromptView.S2Enabled
        Rectangle (0,0 862x24), "%s", text variable: GlobalMessages.gMsgS3.Prompts.topMessage, invisible if: gHMIData.gHideDisplayElementPromptView.S3Enabled
        Rectangle (0,0 862x24), "%s", text variable: GlobalMessages.gMsgS4.Prompts.topMessage, invisible if: gHMIData.gHideDisplayElementPromptView.S4Enabled
        Rectangle (0,0 862x24), "%s", text variable: GlobalMessages.gMsgS5.Prompts.topMessage, invisible if: gHMIData.gHideDisplayElementPromptView.S5Enabled
        Rectangle (0,0 862x24), "%s", text variable: GlobalMessages.gMsgS6.Prompts.topMessage, invisible if: gHMIData.gHideDisplayElementPromptView.S6Enabled
    Rectangle (0,81 1024x31), "Loading Screen...", text list: 'ScreenNames', text index: gHMIData.gScreenNumber
    Rectangle (595,0 166x31), "%s", colour toggle: header.AnyStationFaultHeaderActive, invisible if: NOT header.isAnyFaultState, text list: 'AnyStationAlarmList', text index: header.AnyStationFaultHeader
        p2167032090: header.AnyStationFaultColour
    Group (80,0 861x31)
        Rectangle (0,0 131x31), "%s", text list: 'ModeStatesHeader', text index: header.stationstate
        Rectangle (133,0 133x31), "%s", text list: 'CycleType', text index: header.cycleTypeFeedback
        Rectangle (268,0 97x31), "%s", colour toggle: header.isFaultState, text list: 'FaultState', text index: header.FaultStateHeader
        Rectangle (682,0 147x31), "%s", text list: 'StationNames', text index: header.stationNameSelect
            OnMouseClick: OpenDialog Dialog=dialogStation, OpenModal=True, PositionX=100, PositionY=250
        Rectangle (367,0 147x31), "%s", colour toggle: header.homestateColour, text list: 'HomeState', text index: header.homestate
        Image (830,0 31x31), invisible if: header.flasher, image: FlasherCorner.aus
        Image (830,0 31x31), invisible if: NOT header.flasher, image: FlasherCorner.ein
    Rectangle (595,0 166x31), "%s", colour toggle: header.AnyStationWarningHeaderActive, invisible if: NOT header.isAnyWarningState, text list: 'AnyStationWarningList', text index: header.AnyStationWarningHeader
        p2167032090: header.AnyStationWarningColour
    Rectangle (945,81 76x31), "%d", text variable: gHMIData.gScreenNumber
END_VISUALIZATION

// ---- HMI1/Templates/UnitRow.TcVIS
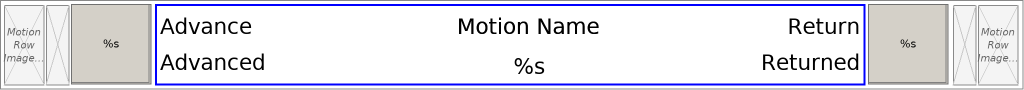
VISUALIZATION UnitRow  // 1024x90
VAR_IN_OUT
	MotionRowInstanceSingle:typeMotionRow; //feedback to motion row to operator
	MotionRowButtonsSingle:typeMotionRowButtons; //button feedback in seperate interface
END_VAR
    Rectangle (155,4 710x81), invisible if: MotionRowInstanceSingle.Returned.bHideCoil AND MotionRowInstanceSingle.bHideName
    Button (868,4 80x80), "%s", text variable: MotionRowInstanceSingle.Returned.NumberOrder, invisible if: MotionRowInstanceSingle.Returned.bHideButton
        tap MotionRowButtonsSingle.btnReturn
        OnMouseDown: execute { gHMIButtons.gAnyButtonPressed := TRUE; }
    Button (71,4 80x80), "%s", text variable: MotionRowInstanceSingle.Advance.NumberOrder, invisible if: MotionRowInstanceSingle.Advance.bHideButton
        tap MotionRowButtonsSingle.btnAdvance
        OnMouseDown: execute { gHMIButtons.gAnyButtonPressed := TRUE; }
    Rectangle (393,50 273x33), "%s", text variable: MotionRowInstanceSingle.strPosn, invisible if: MotionRowInstanceSingle.bHidePosn
    Group (157,10 706x69)
        Rectangle (524,0 182x33), "Return", invisible if: MotionRowInstanceSingle.Returned.bHideCoil or MotionRowInstanceSingle.bIsAbsSymSwitch, text list: 'UnitRowTextText', text index: MotionRowInstanceSingle.IndexLocation + 3, colour variable: MotionRowInstanceSingle.Returned.CoilColour
        Rectangle (235,0 273x33), "Motion Name", invisible if: MotionRowInstanceSingle.bHideName or MotionRowInstanceSingle.bIsAbsSymSwitch, text list: 'UnitRowText', text index: MotionRowInstanceSingle.IndexLocation + 6
        Rectangle (524,36 182x33), "Returned", invisible if: MotionRowInstanceSingle.Returned.bHideDepth or MotionRowInstanceSingle.bIsAbsSymSwitch, text list: 'UnitRowText', text index: MotionRowInstanceSingle.IndexLocation + 4, colour variable: MotionRowInstanceSingle.Returned.FdbkColour
        Rectangle (0,0 207x33), "Advance", text variable: MotionRowInstanceSingle.Advance.valCoil, invisible if: MotionRowInstanceSingle.Advance.bHideCoil or MotionRowInstanceSingle.bIsAbsSymSwitch, text list: 'UnitRowText', text index: MotionRowInstanceSingle.IndexLocation + 0, colour variable: MotionRowInstanceSingle.Advance.CoilColour
        Rectangle (0,36 207x33), "Advanced", invisible if: MotionRowInstanceSingle.Advance.bHideDepth or MotionRowInstanceSingle.bIsAbsSymSwitch, text list: 'UnitRowText', text index: MotionRowInstanceSingle.IndexLocation + 1, colour variable: MotionRowInstanceSingle.Advance.FdbkColour
    Image (4,5 40x80), invisible if: NOT MotionRowInstanceSingle.Advance.InterlockOK OR MotionRowInstanceSingle.Advance.bHideInterlock, image: MotionRowImages.LeftHighlight
    Image (4,5 40x80), invisible if: MotionRowInstanceSingle.Advance.InterlockOK OR MotionRowInstanceSingle.Advance.bHideInterlock, image: MotionRowImages.LeftNot
    Image (978,5 40x80), invisible if: MotionRowInstanceSingle.Returned.InterlockOK OR MotionRowInstanceSingle.Returned.bHideInterlock, image: MotionRowImages.RightNot
    Image (978,5 40x80), invisible if: NOT MotionRowInstanceSingle.Returned.InterlockOK OR MotionRowInstanceSingle.Returned.bHideInterlock, image: MotionRowImages.RightHighlight
    Image (46,5 23x80), invisible if: MotionRowInstanceSingle.Advance.Prompt OR MotionRowInstanceSingle.Advance.bHidePrompt, image: MotionRowImages.PromptNOK
    Image (953,5 23x80), invisible if: NOT MotionRowInstanceSingle.Returned.Prompt OR MotionRowInstanceSingle.Returned.bHidePrompt, image: MotionRowImages.PromptOK
    Image (953,5 23x80), invisible if: MotionRowInstanceSingle.Returned.Prompt OR MotionRowInstanceSingle.Returned.bHidePrompt, image: MotionRowImages.PromptNOK
    Image (46,5 23x80), invisible if: NOT MotionRowInstanceSingle.Advance.Prompt OR MotionRowInstanceSingle.Advance.bHidePrompt, image: MotionRowImages.PromptOK
    Group (157,10 706x69)
        Rectangle (524,0 182x33), "Return", invisible if: MotionRowInstanceSingle.Returned.bHideCoil or NOT MotionRowInstanceSingle.bIsAbsSymSwitch, text list: 'UnitRowText', text index: MotionRowInstanceSingle.IndexLocation + 3 + 10, colour variable: MotionRowInstanceSingle.Returned.CoilColour
        Rectangle (235,0 273x33), "Motion Name", invisible if: MotionRowInstanceSingle.bHideName or NOT MotionRowInstanceSingle.bIsAbsSymSwitch, text list: 'UnitRowText', text index: MotionRowInstanceSingle.IndexLocation + 6 + 10
        Rectangle (524,36 182x33), "Returned", invisible if: MotionRowInstanceSingle.Returned.bHideDepth or NOT MotionRowInstanceSingle.bIsAbsSymSwitch, text list: 'UnitRowText', text index: MotionRowInstanceSingle.IndexLocation + 4 + 10, colour variable: MotionRowInstanceSingle.Returned.FdbkColour
        Rectangle (0,0 207x33), "Advance", text variable: MotionRowInstanceSingle.Advance.valCoil, invisible if: MotionRowInstanceSingle.Advance.bHideCoil or NOT MotionRowInstanceSingle.bIsAbsSymSwitch, text list: 'UnitRowText', text index: MotionRowInstanceSingle.IndexLocation + 0 + 10, colour variable: MotionRowInstanceSingle.Advance.CoilColour
        Rectangle (0,36 207x33), "Advanced", invisible if: MotionRowInstanceSingle.Advance.bHideDepth or NOT MotionRowInstanceSingle.bIsAbsSymSwitch, text list: 'UnitRowText', text index: MotionRowInstanceSingle.IndexLocation + 1 + 10, colour variable: MotionRowInstanceSingle.Advance.FdbkColour
END_VISUALIZATION

// ---- GlobalTextList.TcGTLO
TEXTLIST GlobalTextList
  2452 = ''
  2985 = ' '
  1566 = '            Reject Part?'
  1789 = ' %s Data Entry'
  39 = ' Data Entry'
  2185 = ' Enter Value...'
  962 = ' FB_GetAdaptersInfo'
  2129 = ' FB_GetLicensesEx'
  2732 = ' Integer Entry'
  2906 = ' Reject Part?'
  1685 = ' tDiagScreenPointer %d'
  1493 = ' tDiagScreenPointer %s'
  5065 = '$Row Motion Name + 0'
  2361 = '$Row Motion Name + 1'
  576 = '%5.1f'
  922 = '%5.2f'
  482 = '%5.4f'
  177 = '%5.9f'
  81 = '%d'
  1018 = '%f'
  476 = '%o'
  782 = '%s'
  1224 = '%S'
  485 = '%s %'
  478 = '%s bytes'
  4524 = '%s Data Entry'
  135 = '%s ms'
  2748 = '%s symbols'
  575 = '%s µs'
  667 = '%x'
  1444 = '%X'
  556 = '+0'
  1059 = '+0Memory'
  2991 = '+1'
  225 = '+16'
  97 = '+17'
  1765 = '+24'
  1111 = '+25'
  946 = '+31'
  918 = '+7'
  1494 = '+8'
  1919 = '-1'
  330 = '0'
  459 = '00Slave Number'
  700 = '0Slave Number'
  184 = '1'
  879 = '10'
  1271 = '126'
  1942 = '1262-125'
  888 = '127'
  470 = '16'
  247 = '2'
  1660 = '2-125'
  1462 = '2-1251'
  679 = '255'
  756 = '32'
  1127 = '65535'
  1219 = '8'
  347 = '9999999999'
  1700 = 'AAAA'
  718 = 'Abs/Rel'
  2990 = 'Accelerating'
  2011 = 'ADS'
  6 = 'Advance' | 汉语: '汉语'
  940 = 'Advanced'
  1956 = 'alarm\nview'
  319 = 'alarm text'
  2215 = 'Alarm View'
  606 = 'Alarm View, Machine'
  384 = 'Alarm View, Station 1'
  403 = 'Alarm View, Station 2'
  416 = 'Alarm View, Station 3'
  506 = 'Alarm View, Station 4'
  533 = 'Alarm View, Station 5'
  936 = 'Alarm View, Station 6'
  3612 = 'Alarm Viewq'
  979 = 'Alarms'
  24 = 'AMSid'
  906 = 'AnotherState'
  3273 = 'Apply'
  1284 = 'Are You Sure You Want To Reject The Part?'
  1069 = 'Are you sure you want to reject the part?'
  1315 = 'ASCII'
  200 = 'AUTO\nMODE'
  843 = 'Axis Data'
  3492 = 'Axis Name'
  1230 = 'axis row'
  1781 = 'b0_DiscrapencyErrorInputGroup1'
  2731 = 'b10_DiscrepancyErrorInputGroup3'
  1740 = 'b11_DiscrepancyErrorInputGroup4'
  717 = 'b12_NotUsed'
  768 = 'b13_NotUsed'
  3155 = 'b14_NotUsed'
  3734 = 'b15_NotUsed'
  3183 = 'b1_DiscrapencyErrorInputGroup2'
  622 = 'b2_DiscrapencyErrorInputGroup3'
  2520 = 'b3_DiscrapencyErrorInputGroup4'
  2781 = 'b4_EDMmonitoringErrorEDM1'
  408 = 'b5_EDMmonitoringErrorEDM2'
  1000 = 'b6_NotUsed'
  3066 = 'b7_NotUsed'
  3020 = 'b8_DiscrepancyErrorInputGroup1'
  372 = 'b9_DiscrepancyErrorInputGroup2'
  2888 = 'Back'
  3285 = 'BeckhoffLicence'
  192 = 'BeckhoffPC' | 汉语: '汉语'
  603 = 'BOOT'
  1212 = 'broadcast address'
  2010 = 'Broadcast address. Do not assign'
  4510 = 'Buitton 1'
  3332 = 'CamDataQueued'
  926 = 'CamScalingPending'
  3581 = 'CamTableQueued'
  1604 = 'CamTableQueuued'
  1209 = 'Cancel'
  2419 = 'Channel :%s'
  1780 = 'classic analysis, all in beckhoff twincat3'
  826 = 'CLOSE'
  950 = 'Close'
  1051 = 'CmdBuffered'
  1137 = 'CommsPoCA'
  1330 = 'CommsPorDA'
  1441 = 'CommsPortA'
  780 = 'CommsPortB'
  385 = 'CommsPortC'
  1233 = 'CommsPortD'
  3166 = 'Compensating'
  263 = 'Complexity'
  1496 = 'complexity %s'
  674 = 'Config'
  1377 = 'Config Mode TC'
  46 = 'CONTINUOUS\nCYCLE'
  2770 = 'ContinuousMotion'
  202 = 'Control'
  3305 = 'ControlLoopClosed'
  963 = 'ContstantVelocity'
  1860 = 'Coupled'
  2390 = 'CPU Usage'
  1374 = 'Current Latency'
  1617 = 'Cycle Time'
  844 = 'CycleType'
  785 = 'Cylinder 1'
  481 = 'Data Read NOK'
  1101 = 'Data Read OK'
  3229 = 'Decelerating'
  2015 = 'Default for slaves without aaddress. '
  11 = 'Default for slaves without address. Set electronically to 2-125'
  1289 = 'Demo Licences'
  1774 = 'DemoLicences'
  3573 = 'Depth'
  632 = 'Description'
  246 = 'DeStep[ number'
  161 = 'DeStep[ Step Number'
  510 = 'Device Identificaiton'
  1487 = 'Device Identification'
  1708 = 'Device Infomation'
  868 = 'Disabled'
  3627 = 'DiscreteMotion'
  640 = 'Down'
  2466 = 'DriveDeviceError'
  1534 = 'DriveLimitActive'
  839 = 'DRY\nCYCLE'
  2893 = 'Edit'
  149 = 'ENABLE\nPENDANT'
  631 = 'ENABLE\nREMOTE\nCONTROL'
  593 = 'ENABLE BENDANT'
  3484 = 'Enter a value...'
  1975 = 'Error'
  1556 = 'ErrorID'
  983 = 'ErrorPropagationDelayed'
  2486 = 'ErrorStop'
  684 = 'EtherCAT'
  454 = 'EtherCAT\nDiagnostics'
  338 = 'EtherCAT Clave Details'
  513 = 'EtherCAT Detailed Slave Details'
  1332 = 'EtherCAT Diagnostics'
  1412 = 'EtherCAT Slave Details'
  255 = 'EtherCAT Slave ID:\n %d'
  645 = 'EtherCAT Slave ID: %d'
  151 = 'EtherCATDongle' | 汉语: '汉语'
  1669 = 'ExpirationTime'
  427 = 'ExternalLatchValid'
  990 = 'ExtSetPointGenEnabled'
  2952 = 'Failed Licences'
  840 = 'Fault'
  1555 = 'Fault Locaiton'
  462 = 'Fault Location'
  852 = 'FaultState'
  2089 = 'FB_GetDeviceIdentificationEx'
  1670 = 'FB_GetLicensesEx'
  520 = 'FFFFFFFF'
  1203 = 'FFFFFFFFF'
  3850 = 'french'
  447 = 'GATE 1\nACCESS \n REQUEST'
  707 = 'GATE 1\nACCESS REQUEST'
  869 = 'GATE 1 ACCESS REQUEST'
  181 = 'GATE 2\nACCESS \n REQUEST'
  3447 = 'GenDevTypeLic'
  3752 = 'german'
  805 = 'gmsgTest.msgHeader.col1'
  942 = 'GroupBox'
  1663 = 'gSafetyCPUADSadr'
  2884 = 'gSafetyCPUState'
  3901 = 'gSafetyProgramChecksum'
  2328 = 'gSafetySerialNumber'
  2962 = 'HadJob'
  2696 = 'HardwareCPU'
  2291 = 'HardwareDate'
  578 = 'HardwareModel'
  434 = 'HardwareSerialNo'
  2603 = 'HardwareVersion'
  3230 = 'HasBeenStopped'
  3108 = 'HasJob'
  1106 = 'Help'
  1768 = 'Hex'
  57 = 'HEX'
  240 = 'HEX/DEC'
  580 = 'HMI\nSystem'
  614 = 'HMI System'
  709 = 'Homed'
  67 = 'HomeState'
  3520 = 'Homing'
  1944 = 'HomingBusy'
  1156 = 'Hostname'
  539 = 'I'
  4091 = 'iAccessGate1Diag'
  4248 = 'iAccessGate2Diag'
  1049 = 'iEnablePendantSafetyDevicesuint'
  3271 = 'iEnableSafetyDevicesuint'
  4412 = 'iEnablingPendantDiag'
  1625 = 'iEstop1Diag'
  258 = 'iEstop2Diag'
  1803 = 'iEstop3Diag'
  3554 = 'iGroupPort_ErrAck'
  889 = 'ImageDevice'
  1513 = 'ImageLevel'
  104 = 'ImageOSName'
  1252 = 'ImageOsName'
  2966 = 'ImageOsVersion'
  136 = 'ImageVersion'
  1056 = 'iModuleFault'
  1068 = 'INIT'
  1390 = 'InitError'
  3745 = 'InPositionArea'
  3366 = 'InTargetPosition'
  1517 = 'INTEL'
  393 = 'Invalid Licences'
  272 = 'InvalidVendor'
  2377 = 'IoDataInvalid'
  1972 = 'IoDataInvalidf'
  4538 = 'iResetFBs'
  1512 = 'iRunStop'
  605 = 'k'
  129 = 'L'
  1834 = 'Label'
  1047 = 'lang row'
  85 = 'langauge row'
  141 = 'langauge row abs'
  710 = 'Language'
  767 = 'language row'
  941 = 'Last Operation'
  748 = 'LicenceID'
  694 = 'LicenceIdLabel'
  2654 = 'LicenceIdLicenceIdLabel'
  1938 = 'LicenceName'
  2136 = 'Loading Screen...'
  626 = 'Location'
  677 = 'LOCK \nACCESS \nGATE'
  887 = 'LOCK ACCESS GATE'
  1134 = 'M'
  335 = 'Machine\nLayout'
  479 = 'MachineSettings.Setting[INDEX].TextNamedd'
  910 = 'Main\nMenu'
  564 = 'Manual\nAxis\nMotion'
  150 = 'MANUAL\nMODE'
  566 = 'Manual\nMotions'
  1483 = 'Max Latency'
  1386 = 'MaxCount'
  1739 = 'Memory'
  1307 = 'Memory\nView'
  2002 = 'Memory Location'
  1017 = 'MemoryMemory Location'
  3103 = 'Menu 1'
  2056 = 'Menu 2'
  1966 = 'Menu 3'
  4851 = 'Menu 4'
  4054 = 'Menu 5'
  2436 = 'Menu Buitton 1'
  599 = 'Menu Button 1'
  1574 = 'Menu Button 2'
  2217 = 'Menu Button 3'
  2986 = 'Menu Button 4'
  646 = 'Menu Button 5'
  1339 = 'Message'
  132 = 'Message Message '
  623 = 'Message Message Message Message Message Message Message Message Message Message '
  1491 = 'Message Text'
  344 = 'Mode'
  4343 = 'Mode Rows'
  3602 = 'Mode Screen Motion View'
  655 = 'Motion Name'
  2407 = 'MotionCommandsLocked'
  557 = 'MotionState'
  612 = 'MOTO'
  3831 = 'Moving'
  697 = 'MsgTe'
  1354 = 'msgtest. '
  3488 = 'Multi-Ordinal Step'
  3649 = 'NcApplicationRequest'
  2751 = 'NcCycleCounter'
  1027 = 'nDevType'
  1375 = 'NegativeDirection'
  1223 = 'NetID: %s'
  610 = 'NewTargetPosition'
  683 = 'Next'
  390 = 'Next Page\nV'
  2091 = 'Next Row'
  4369 = 'Next Step'
  1867 = 'Nextg'
  2073 = 'No'
  124 = 'NOK To Build' | 汉语: '汉语'
  932 = 'NoState'
  1786 = 'NotMoving'
  714 = 'num'
  907 = 'Number Rejects'
  140 = 'OEM Licences' | 汉语: '汉语'
  1575 = 'OemLicence'
  639 = 'of %d'
  636 = 'OK'
  886 = 'OK to Build'
  471 = 'OK To Build'
  3052 = 'Old Value'
  503 = 'OP'
  1128 = 'Operational'
  3859 = 'OpMode'
  435 = 'OptInfo'
  1346 = 'Over Cycle Time!'
  802 = 'Page %d'
  99 = 'Part'
  1026 = 'Part Description'
  583 = 'Part Present'
  925 = 'Pending Licences'
  218 = 'PendingLicences'
  1954 = 'PhasingActive'
  1080 = 'Platern ID'
  799 = 'Platern Number Ops'
  939 = 'PLC High Record Scan'
  693 = 'PLC High Scan Record'
  915 = 'PLC Scan Number'
  604 = 'PLC Scan Time'
  630 = 'PLC Scan Time Actual'
  52 = 'PLC Scan Time Record'
  14 = 'PLC Scan Time Record Scan'
  122 = 'PLC Scan Time Requested' | 汉语: '汉语'
  1619 = 'PLC_ReadSymInfo'
  1589 = 'Port: %s'
  504 = 'portA'
  484 = 'PortA'
  1584 = 'PortB'
  1033 = 'PortC'
  1690 = 'PositiveDirection'
  696 = 'POWER\nOFF'
  981 = 'POWER\nON'
  270 = 'PREOP'
  1800 = 'Previous'
  708 = 'productCode'
  1544 = 'Profibus DP\nDiagnopstics'
  1235 = 'Profibus DP\nDiagnostics'
  1600 = 'Profibus DP Slave Help'
  721 = 'Profibus/DP'
  1750 = 'Profibus/DP\nDiagnostics'
  188 = 'PROFINET Detailed Slave Details'
  205 = 'PROFINET/PN'
  3659 = 'Program Version'
  457 = 'Programming Tool, Master or Slave aAddress'
  176 = 'Programming Tool, master or slave address'
  414 = 'Prompt View, Station 1'
  921 = 'Prompt View, Station 2'
  711 = 'Prompt View, Station 3'
  854 = 'Prompt View, Station 4'
  755 = 'Prompt View, Station 5'
  699 = 'Prompt View, Station 6'
  1881 = 'ProtectedMode'
  3521 = 'PTPmode'
  2257 = 'Q'
  4298 = 'qComError'
  3063 = 'qCommStartup'
  3221 = 'qFBDeactive'
  3102 = 'qFBError'
  4488 = 'qInRun'
  2545 = 'qOtherError'
  1552 = 'qOutError'
  3228 = 'qRun'
  235 = 'Quarantine Part'
  3193 = 'Read'
  2255 = 'REAL'
  2368 = 'Reject'
  1841 = 'Reject Part?'
  1518 = 'Request'
  654 = 'Requestel'
  728 = 'Reset'
  2806 = 'Restart'
  2369 = 'Restart TC'
  2688 = 'Restriction'
  2488 = 'Result'
  795 = 'Return'
  276 = 'RETURN\nHOME'
  236 = 'Returned'
  841 = 'Returnn'
  873 = 'revisionNo'
  4077 = 'Row'
  301 = 'Row Motion Name'
  4451 = 'Row Motion Name + 0'
  2003 = 'Row Motion Name + 1'
  1745 = 's'
  1073 = 'SAFEOP'
  256 = 'Scrap Part'
  808 = 'Screen Name'
  491 = 'sd '
  989 = 'sdsd'
  2575 = 'sdsdLicenceIdLicenceIdLabel'
  1542 = 'Second'
  766 = 'SELECT ALL'
  837 = 'SEMI'
  425 = 'SEMI-AUTO\nMODE'
  4568 = 'Sequence\nSetup'
  3735 = 'Sequence Setup'
  624 = 'Serial Number Valid'
  783 = 'Serial Valid'
  1399 = 'SerialNo'
  1760 = 'Setting'
  3666 = 'Setting Name'
  72 = 'sExpirationTime'
  1782 = 'SIEMENS/754'
  765 = 'SILENCE\nHORN'
  818 = 'SINGLE\n CYCLE'
  83 = 'SINGLE CYCLE' | 汉语: '汉语'
  198 = 'Slave Number' | 汉语: '汉语'
  982 = 'SlaveDisabled'
  65 = 'SlaveNotPresent'
  538 = 'SlaveSigfnalsLinkError'
  819 = 'SlaveSignalsError'
  162 = 'SlaveSignalsLinkError'
  103 = 'SlaveSignalsMissingLink'
  250 = 'SlaveSignasError'
  815 = 'sName           '
  2740 = 'SoftLimitMaxExceeded'
  3564 = 'SoftLimitMinExceeded'
  3478 = 'spare'
  2162 = 'special\nmessage'
  1427 = 'Special Address used by Class 2 Master or FieldPG setting device'
  1394 = 'ss'
  1095 = 'StandStill'
  905 = 'START\nAUTO\nCYCLE'
  466 = 'START AUTO CYCLE'
  251 = 'STARTAUTO CYCLE'
  814 = 'StationName'
  7 = 'StationState' | 汉语: '汉语'
  3355 = 'Status'
  2052 = 'Step'
  4459 = 'Step Number'
  1484 = 'Stop'
  746 = 'STOP\nAUTO\nCYCLE'
  252 = 'STOP\nEOC'
  635 = 'STOP END\nOF CYCLE'
  1783 = 'Stop TC'
  1148 = 'Stopping'
  472 = 'sType'
  1146 = 'sType          '
  3971 = 'ST_AxisStatus'
  1581 = 'ST_EcCrcError'
  1634 = 'ST_EcSlaveConfigData'
  1554 = 'ST_EcSlaveIdentity'
  2008 = 'Swap 1'
  961 = 'Syb/Rel'
  754 = 'Sym/Abs'
  53 = 'SYMCOUNT'
  2510 = 'SYMSIZE'
  3596 = 'SynchronizedMotion'
  1366 = 'Target'
  2172 = 'TargetType'
  701 = 'Task Name'
  668 = 'TC Mode'
  2788 = 'TC Restart'
  1844 = 'TC_CpuUsage'
  2145 = 'TC_SysLatency'
  230 = 'tDiagScreenSize %d'
  1070 = 'tDiagScreenSize %s'
  1263 = 'tDiagScreenWidth %d'
  74 = 'tDiagScreenWidth %s'
  877 = 'test12'
  2059 = 'tExpirationTime'
  812 = 'the time'
  514 = "Thomas O'Kane"
  2046 = 'Time Raised'
  1482 = 'Time Resolved'
  945 = 'Top Header'
  1055 = 'TwinCATBuild'
  1175 = 'TwinCATLevel'
  1961 = 'TwinCATRevision'
  60 = 'TwinCATVersion'
  4123 = 'TwinSAFE\nStatus'
  4648 = 'TwinSAFE Runtime 1'
  4055 = 'typeSeqRow'
  1151 = 'Typical master or slaves '
  786 = 'Unit Name'
  277 = 'Units'
  1679 = 'Up'
  1976 = 'Update'
  2305 = 'UpdateCycleTimed'
  1678 = 'UpdateCycleTimedd'
  784 = 'UpdateTaskIndex'
  3452 = 'USBDongle'
  1798 = 'UsedCount'
  3898 = 'User Program'
  980 = 'V'
  282 = 'V%s'
  451 = 'Valid Licences'
  199 = 'ValidLicences'
  1906 = 'Value'
  413 = 'VendorID'
  163 = 'Version'
  392 = 'VolumeNo'
  512 = 'Warning'
  253 = 'Warning View, Machine'
  407 = 'Warning View, Station 1'
  690 = 'Warning View, Station 2'
  872 = 'Warning View, Station 3'
  110 = 'Warning View, Station 4'
  954 = 'Warning View, Station 5'
  133 = 'Warning View, Station 6'
  25 = 'Warnings'
  1532 = 'WIP'
  2645 = 'Write'
  473 = 'x'
  2862 = 'X'
  241 = '^'
  8 = '^\nPrevious Page'
  275 = '^?'
  2662 = '汉语'
END_TEXTLIST

// ---- HMI1/Data/CycleType.TcTLO
TEXTLIST CycleType
  0 = ' '
  1 = 'Continuous Cycle' | 汉语: '汉语'
  2 = 'Single Cycle' | 汉语: '汉语'
  3 = 'other state' | 汉语: '汉语'
   = ''
END_TEXTLIST

// ---- HMI1/Data/FaultState.TcTLO
TEXTLIST FaultState
  0 = ' '
  1 = 'Fault' | 汉语: '汉语'
   = ''
END_TEXTLIST

// ---- HMI1/Data/HomeState.TcTLO
TEXTLIST HomeState
  0 = 'Not Home' | 汉语: '汉语'
  1 = 'Homing' | 汉语: '汉语'
  2 = 'Home' | 汉语: '汉语'
   = ''
END_TEXTLIST

// ---- HMI1/Data/ModeStates.TcTLO
TEXTLIST ModeStates
  0 = 'No State' | 汉语: '汉语'
  1 = 'Power Off' | 汉语: '汉语'
  2 = 'Power On' | 汉语: '汉语'
  3 = 'Manual Mode' | 汉语: '汉语'
  4 = 'Auto Mode' | 汉语: '汉语'
  5 = 'Auto Cycling' | 汉语: '汉语'
  6 = 'Semi Auto'
  7 = 'Fault'
  8 = 'Bypass'
  9 = 'Auto Cycle Stopping'
  10 = 'Dry Cycle'
   = ''
END_TEXTLIST

// ---- HMI1/Data/ModeStatesHeader.TcTLO
TEXTLIST ModeStatesHeader
  0 = 'No State' | 汉语: '汉语'
  1 = 'Power Off' | 汉语: '汉语'
  2 = 'Power On' | 汉语: '汉语'
  3 = 'Manual' | 汉语: '汉语'
  4 = 'Auto'
  5 = 'Auto Cycle'
  6 = 'Semi Auto'
  7 = 'Fault'
  8 = 'Bypass'
  9 = 'Stopping'
  10 = 'State2'
   = ''
END_TEXTLIST

